TYPE ST_DS_Parameter :
STRUCT
	Druck_Max	: REAL;
	Druck_Min	: REAL;
END_STRUCT
END_TYPE

(* stored: Version 1.1.0.1, ProductVersion 3.1.4024.9
   DUT ST_DS_Parameter: Id {5e91c0cd-ddfe-48dd-9827-ec56d8b8420d} *)
